// TIA Portal V18 export
// export: Created 2026-03-12T16:04:34.3424017Z, ExportSetting WithDefaults, DisplayName Totally Integrated Automation Portal, DisplayVersion V18 Update 5, DisplayName TIA Portal Openness, DisplayVersion V18 Update 5, DisplayName TIA Portal Version Control Interface, DisplayVersion V18, DisplayName SINAMICS Startdrive Advanced, DisplayVersion V18, DisplayName SINAMICS Startdrive G130, G150, S120, S150, SINAMICS MV, S210, DisplayVersion V18, DisplayName SINAMICS Startdrive G110M, G120, G120C, G120D, G120P, G115D, DisplayVersion V18, DisplayName STEP 7 Professional, DisplayVersion V18 Update 5, DisplayName STEP 7 Safety, DisplayVersion V18, DisplayName WinCC Professional, DisplayVersion V18 Update 5
FUNCTION_BLOCK "FB BITS TO DOUBLE WORD"   // FB5, SCL
{ S7_Optimized_Access := 'TRUE' }
VERSION : 0.1
// stored: AutoNumber true, IsIECCheckEnabled false, IsRetainMemResEnabled false, MemoryReserve 100, SetENOAutomatically false, UDAEnableTagReadback false
   VAR_INPUT
      SIGNAL_Bit0 : Bool;   // Sinal de entrada 1
      SIGNAL_Bit1 : Bool;   // Sinal de entrada 2
      SIGNAL_Bit2 : Bool;   // Sinal de entrada 3
      SIGNAL_Bit3 : Bool;   // Sinal de entrada 4
      SIGNAL_Bit4 : Bool;   // Sinal de entrada 5
      SIGNAL_Bit5 : Bool;   // Sinal de entrada 6
      SIGNAL_Bit6 : Bool;   // Sinal de entrada 7
      SIGNAL_Bit7 : Bool;   // Sinal de entrada 8
      SIGNAL_Bit8 : Bool;   // Sinal de entrada 9
      SIGNAL_Bit9 : Bool;   // Sinal de entrada 10
      SIGNAL_Bit10 : Bool;   // Sinal de entrada 11
      SIGNAL_Bit11 : Bool;   // Sinal de entrada 12
      SIGNAL_Bit12 : Bool;   // Sinal de entrada 13
      SIGNAL_Bit13 : Bool;   // Sinal de entrada 14
      SIGNAL_Bit14 : Bool;   // Sinal de entrada 15
      SIGNAL_Bit15 : Bool;   // Sinal de entrada 16
      SIGNAL_Bit16 : Bool;   // Sinal de entrada 17
      SIGNAL_Bit17 : Bool;   // Sinal de entrada 18
      SIGNAL_Bit18 : Bool;   // Sinal de entrada 19
      SIGNAL_Bit19 : Bool;   // Sinal de entrada 20
      SIGNAL_Bit20 : Bool;   // Sinal de entrada 21
      SIGNAL_Bit21 : Bool;   // Sinal de entrada 22
      SIGNAL_Bit22 : Bool;   // Sinal de entrada 23
      SIGNAL_Bit23 : Bool;   // Sinal de entrada 24
      SIGNAL_Bit24 : Bool;   // Sinal de entrada 25
      SIGNAL_Bit25 : Bool;   // Sinal de entrada 26
      SIGNAL_Bit26 : Bool;   // Sinal de entrada 27
      SIGNAL_Bit27 : Bool;   // Sinal de entrada 28
      SIGNAL_Bit28 : Bool;   // Sinal de entrada 29
      SIGNAL_Bit29 : Bool;   // Sinal de entrada 30
      SIGNAL_Bit30 : Bool;   // Sinal de entrada 31
      SIGNAL_Bit31 : Bool;   // Sinal de entrada 32
   END_VAR
   VAR_OUTPUT
      BITS_TO_DWORD : DWord;   // Word de saída com os sinais montados
   END_VAR
BEGIN
   // Word Alarmes - Montando bits em uma double word

   // Bits recebidos de campo
   #"BITS_TO_DWORD".%X0 := #SIGNAL_Bit0;
   #"BITS_TO_DWORD".%X1 := #SIGNAL_Bit1;
   #"BITS_TO_DWORD".%X2 := #SIGNAL_Bit2;
   #"BITS_TO_DWORD".%X3 := #SIGNAL_Bit3;
   #"BITS_TO_DWORD".%X4 := #SIGNAL_Bit4;
   #"BITS_TO_DWORD".%X5 := #SIGNAL_Bit5;
   #"BITS_TO_DWORD".%X6 := #SIGNAL_Bit6;
   #"BITS_TO_DWORD".%X7 := #SIGNAL_Bit7;
   #"BITS_TO_DWORD".%X8 := #SIGNAL_Bit8;
   #"BITS_TO_DWORD".%X9 := #SIGNAL_Bit9;
   #"BITS_TO_DWORD".%X10 := #SIGNAL_Bit10;
   #"BITS_TO_DWORD".%X11 := #SIGNAL_Bit11;
   #"BITS_TO_DWORD".%X12 := #SIGNAL_Bit12;
   #"BITS_TO_DWORD".%X13 := #SIGNAL_Bit13;
   #"BITS_TO_DWORD".%X14 := #SIGNAL_Bit14;
   #"BITS_TO_DWORD".%X15 := #SIGNAL_Bit15;
   #"BITS_TO_DWORD".%X16 := #SIGNAL_Bit16;
   #"BITS_TO_DWORD".%X17 := #SIGNAL_Bit17;
   #"BITS_TO_DWORD".%X18 := #SIGNAL_Bit18;
   #"BITS_TO_DWORD".%X19 := #SIGNAL_Bit19;
   #"BITS_TO_DWORD".%X20 := #SIGNAL_Bit20;
   #"BITS_TO_DWORD".%X21 := #SIGNAL_Bit21;
   #"BITS_TO_DWORD".%X22 := #SIGNAL_Bit22;
   #"BITS_TO_DWORD".%X23 := #SIGNAL_Bit23;
   #"BITS_TO_DWORD".%X24 := #SIGNAL_Bit24;
   #"BITS_TO_DWORD".%X25 := #SIGNAL_Bit25;
   #"BITS_TO_DWORD".%X26 := #SIGNAL_Bit26;
   #"BITS_TO_DWORD".%X27 := #SIGNAL_Bit27;
   #"BITS_TO_DWORD".%X28 := #SIGNAL_Bit28;
   #"BITS_TO_DWORD".%X29 := #SIGNAL_Bit29;
   #"BITS_TO_DWORD".%X30 := #SIGNAL_Bit30;
   #"BITS_TO_DWORD".%X31 := #SIGNAL_Bit31;
END_FUNCTION_BLOCK
